{attribute 'qualified_only'}
{attribute 'to_string'}
TYPE E_LinearActuatorHomingStates :
(
	Idle:=0,
	CheckIfEnabled,
	EnableAxis1,
	EnableAxis2,
	ResetAxis1,
	ResetAxis2,
	MoveToTop,
	WaitingForHalt,
	SettingHomePos,
	DisableAxis,
	WrapUp
)UINT := Idle
;
END_TYPE

(* stored: Version 1.1.0.1, ProductVersion 3.1.4024.12
   EnumerationTextList E_LinearActuatorHomingStates: Id {37d6df4a-905b-4439-8b8b-d421c3f0e37d} *)
